// TIA Portal V18 export
// export: Created 2026-06-21T12:15:02Z, ExportSetting WithDefaults
PlcWatchTable "WT_PLC1_Fake_PLC2_Modbus_Return"
  PlcWatchTableEntry ""DB_PLC1_Recv_From_PLC2_DB".AckSeq"
  PlcWatchTableEntry ""DB_PLC1_Recv_From_PLC2_DB".Done_Branch2"
  PlcWatchTableEntry ""DB_PLC1_Recv_From_PLC2_DB".Done_Discharge2"
  PlcWatchTableEntry ""DB_PLC1_Recv_From_PLC2_DB".Done_Recipe"
  PlcWatchTableEntry ""DB_PLC1_Recv_From_PLC2_DB".Alarm"
  PlcWatchTableEntry ""DB_PLC1_Recv_From_PLC2_DB".State"
  PlcWatchTableEntry ""DB_PLC1_Recv_From_PLC2_DB".PID_Bon4_SP"
  PlcWatchTableEntry ""DB_PLC1_Recv_From_PLC2_DB".PID_Bon4_PV"
  PlcWatchTableEntry ""DB_PLC1_Recv_From_PLC2_DB".PID_Bon4_CV"
  PlcWatchTableEntry ""DB_PLC1_Recv_From_PLC2_DB".Heartbeat"
